// TwinCAT 3 PLC project Untitled1
// ProgramVersion: 3.1.4023.0
// libraries:
//   Tc2_Standard, * (Beckhoff Automation GmbH)
//   Tc2_System, * (Beckhoff Automation GmbH)
//   Tc3_Module, * (Beckhoff Automation GmbH)
// project tree:
//   / PlcTask.TcTTO (not stored)
//   POUs/ MAIN.TcPOU
//   TASK1/ G_Task1.TcGVL (not stored), P_Task1.TcPOU, SensorBrand.TcDUT
//   TASK2/ G_Task2.TcGVL, P_Task2.TcPOU, ST_Timer.TcDUT

// ---- TASK1/SensorBrand.TcDUT

TYPE SensorBrand :
(
	Sick:= 0,
	Pilz:=1,
	Parker:=2,
	Bosch:=3
	
	
);
END_TYPE

// ---- TASK2/ST_Timer.TcDUT
TYPE ST_Timer :
STRUCT
	
END_STRUCT
END_TYPE

// ---- TASK2/G_Task2.TcGVL
{attribute 'qualified_only'}
VAR_GLOBAL
END_VAR

// ---- POUs/MAIN.TcPOU
PROGRAM MAIN
VAR
	
END_VAR

P_Task1();
P_task2();

END_PROGRAM

// ---- TASK1/P_Task1.TcPOU
PROGRAM P_Task1
VAR
	pPointer:POINTER TO DATE_AND_TIME;
	tRef:REFERENCE TO TIME REF=G_Task1.tTid;
	fbTon : TON ;
	
	
	
END_VAR

pPointer:=ADR(G_Task1.dtvariable);
pPointer^ :=DT#2023-02-10-15:31:19;

tRef  :=T#10S;
G_Task1.aDatoArray[3]:=D#2023-02-25;
G_Task1.eSensor1:=SensorBrand.Parker;
fbTon(
		IN:=G_Task1.bTimerStart,
		PT:=G_Task1.tTimer,
		ET=>G_Task1.tEllapsedTime,
		Q=>G_Task1.bTimerOn

);

END_PROGRAM

// ---- TASK2/P_Task2.TcPOU
PROGRAM P_Task2
VAR
END_VAR

END_PROGRAM
